TYPE ST_GZ_Zustand :
STRUCT
	AktuellesVolummen	: REAL;
	Durchfluss			: REAL;
	Freigabe			: BOOL;
	Temperatur			: REAL;
END_STRUCT
END_TYPE

(* stored: Version 1.1.0.1, ProductVersion 3.1.4024.9
   DUT ST_GZ_Zustand: Id {2cb0f778-3b65-4e96-b898-20cbb758298c} *)
